SUBAPPLICATION mapping (* Subapplication Type *)
  (* Standard: 61499-2 *)
  (* Version 1.0, 2023-07-15, franz *)
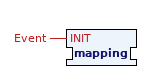
  EVENT_INPUT
    INIT;
  END_EVENT
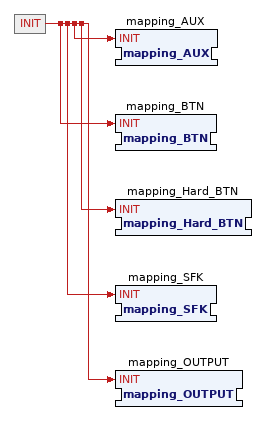
  SUBAPPS
    mapping_BTN : mapping_BTN;
    mapping_SFK : mapping_SFK;
    mapping_AUX : mapping_AUX;
    mapping_Hard_BTN : mapping_Hard_BTN;
    mapping_OUTPUT : mapping_OUTPUT;
  END_SUBAPPS
  EVENT_CONNECTIONS
    INIT TO mapping_BTN.INIT;
    INIT TO mapping_SFK.INIT;
    INIT TO mapping_AUX.INIT;
    INIT TO mapping_Hard_BTN.INIT;
    INIT TO mapping_OUTPUT.INIT;
  END_CONNECTIONS
END_SUBAPPLICATION
